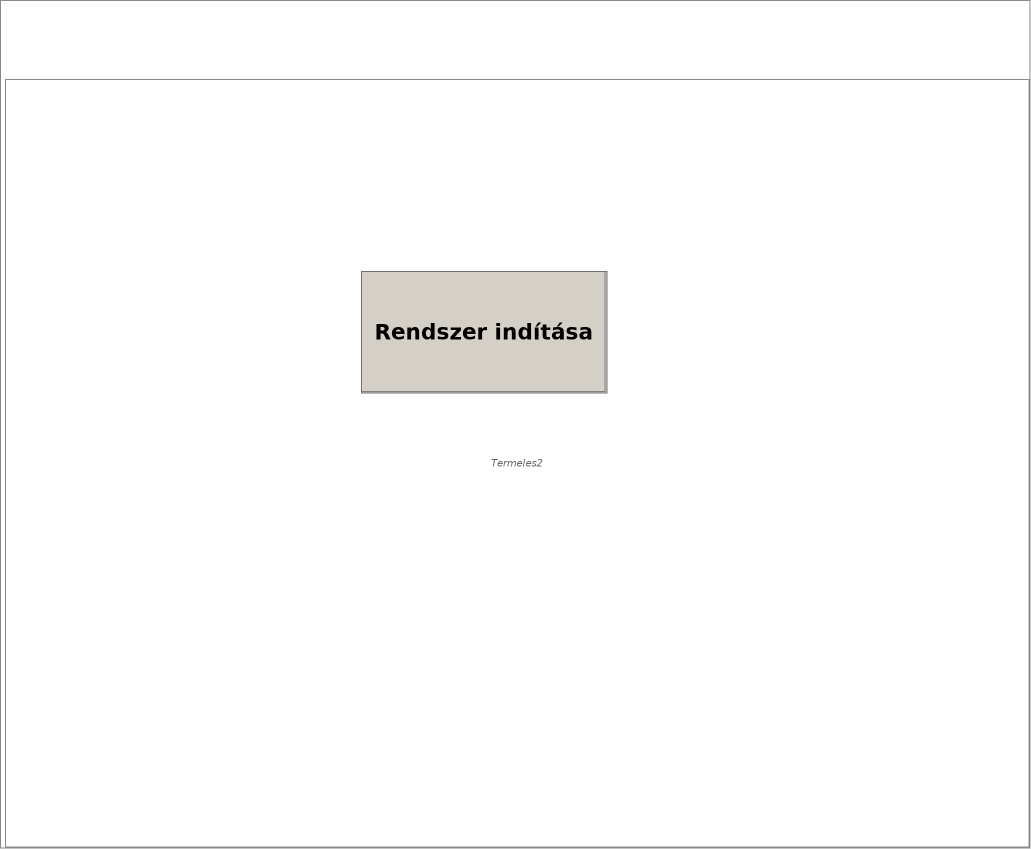
VISUALIZATION Visualization2  // 1031x849
    TabControl (5,79 1024x768), invisible if: GVL.bSystemNotStarted, input disabled if: GVL.bSystemNotStarted
        shows Termeles2()
        shows TempZoli()
        shows TempRobot()
        shows TempJozsi()
        shows TempPisti()
        shows Laser()
        shows HegesztesGrafikon()
        [0]: TabTitle=Termelés
        [1]: TabTitle=Főnök
        [2]: TabTitle=Robot
        [3]: TabTitle=Józsi
        [4]: TabTitle=Pisti
        [5]: TabTitle=Lézer
        [6]: TabTitle=Útmérés
    Button (361,271 246x122), "Rendszer indítása", invisible if: GVL.bSystemStarted, input disabled if: GVL.bSystemStarted
        OnMouseClick: execute { INIT.iState:=1; }
END_VISUALIZATION

(* stored: Version 1.1.0.1, ProductVersion 3.1.4024.11
   Visu Visualization2: Id {f9cbb580-02c2-4cbd-93d7-299cb9ed791f} *)
